(* Logix 5000 project; controller SX_V040001_C001 vendor 1 type 14 code 77 rev 16.23; software revision 16.04; part 35 of 35 *)
(* tags used below, declared in another part *)
   testRick : BOOL;
   Basic : INT;
   G_AOutput : DINT[8];
   G_DOutput : DINT[3];
(* MainProgram, continued *)

ROUTINE WriteOutput   (* ladder *)
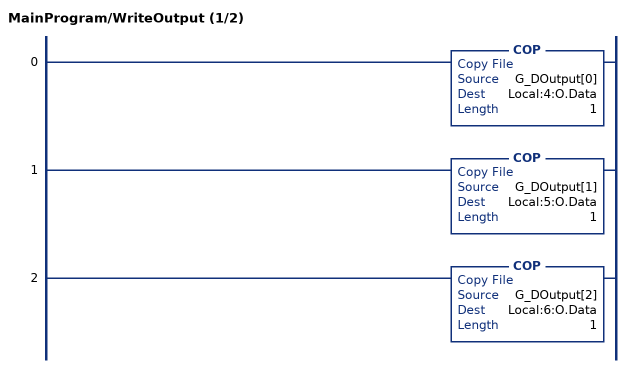
   0: COP(G_DOutput[0],Local:4:O.Data,1);
   1: COP(G_DOutput[1],Local:5:O.Data,1);
   2: COP(G_DOutput[2],Local:6:O.Data,1);
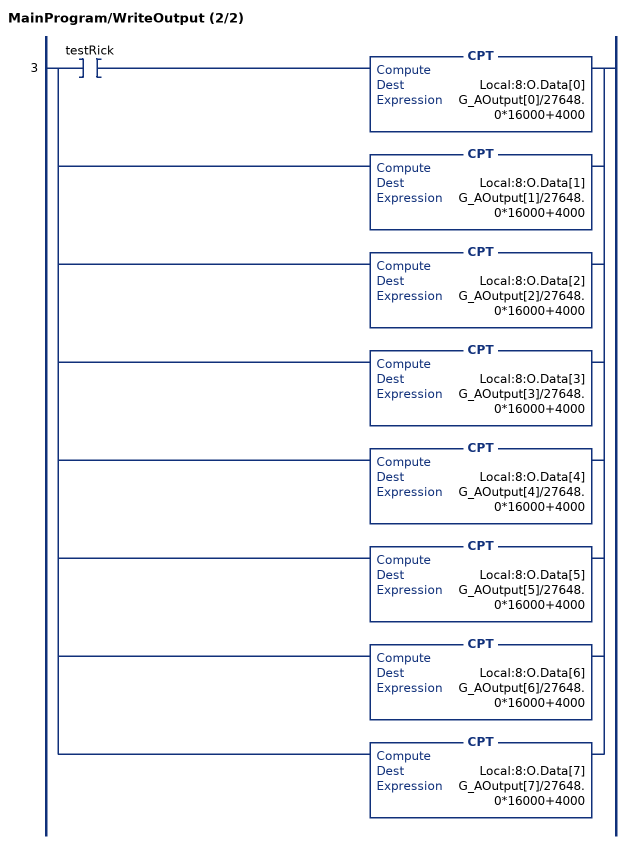
   3: [XIC(testRick) CPT(Local:8:O.Data[0],G_AOutput[0]/27648.0*16000+4000) ,CPT(Local:8:O.Data[1],G_AOutput[1]/27648.0*16000+4000) ,CPT(Local:8:O.Data[2],G_AOutput[2]/27648.0*16000+4000) ,CPT(Local:8:O.Data[3],G_AOutput[3]/27648.0*16000+4000) ,CPT(Local:8:O.Data[4],G_AOutput[4]/27648.0*16000+4000) ,CPT(Local:8:O.Data[5],G_AOutput[5]/27648.0*16000+4000) ,CPT(Local:8:O.Data[6],G_AOutput[6]/27648.0*16000+4000) ,CPT(Local:8:O.Data[7],G_AOutput[7]/27648.0*16000+4000) ];
END_ROUTINE
END_PROGRAM

PROGRAM Tastk_100MS   (* main routine Task_100MS *)

ROUTINE Task_100MS   (* ladder *)
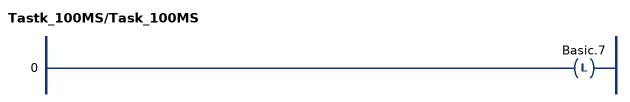
   0: OTL(Basic.7);
END_ROUTINE
END_PROGRAM
